FUNCTION_BLOCK FB_Cylinder 
VAR_INPUT
END_VAR
VAR_OUTPUT
	bExtended : BOOL;
END_VAR
VAR
	bStart AT%Q* : BOOL;
	fbExtendedSignal : BoolIn;
END_VAR

bExtended := fbExtendedSignal.getValue;

END_FUNCTION_BLOCK

(* stored: Version 1.1.0.1, ProductVersion 3.1.4024.0
   POU FB_Cylinder: Id {4dff6417-8bf1-4724-a444-43bb6b5867e9}, SpecialFunc None *)
